Universal Robots URScript: test1.script

def unnamed():
  global _hidden_verificationVariable=0
  set_tcp(p[0.0,0.0,0.0,0.0,0.0,0.0])
  set_safety_mode_transition_hardness(1)
  set_gravity([0.0, 0.0, 9.82])
  set_tool_communication(False, 115200, 0, 1, 1.5, 3.5)
  set_tool_output_mode(0)
  set_tool_digital_output_mode(0, 1)
  set_tool_digital_output_mode(1, 1)
  set_tool_voltage(0)
  set_target_payload(0.000000, [0.000000, 0.000000, 0.000000], [0.000000, 0.000000, 0.000000, 0.000000, 0.000000, 0.000000])
  set_standard_analog_input_domain(0, 1)
  set_standard_analog_input_domain(1, 1)
  set_tool_analog_input_domain(0, 1)
  set_tool_analog_input_domain(1, 1)
  set_analog_outputdomain(0, 0)
  set_analog_outputdomain(1, 0)
  set_input_actions_to_default()
  # begin: URCap Installation Node
  #   Source: External Control, 1.0.5, FZI Research Center for Information Technology
  #   Type: External Control
  # end: URCap Installation Node
  step_count_bf1d607d_5cad_4ca6_951d_d38089d2c4e9 = 0.0
  thread Step_Counter_Thread_272bec76_1d24_4e5e_b286_867ec8d2c18c():
    while (True):
      step_count_bf1d607d_5cad_4ca6_951d_d38089d2c4e9 = step_count_bf1d607d_5cad_4ca6_951d_d38089d2c4e9 + 1.0
      sync()
    end
  end
  run Step_Counter_Thread_272bec76_1d24_4e5e_b286_867ec8d2c18c()
  global Waypoint_1_p=p[.365377612465, -.462828783151, .512939210108, -1.170877947002, 2.833532311999, .102825613587]
  global Waypoint_1_q=[-0.6912114986220512, -1.7813268732349261, -1.267368403083033, -1.6883155612163208, 1.667533326914021, 0.09468801413845322]
  global Waypoint_2_p=p[.000000000000, -.232900000168, 1.079399999952, -.000000000000, 2.221441469307, -2.221441468851]
  global Waypoint_2_q=[0.0, -1.5707963267948966, 0.0, -1.5707963267948974, 0.0, 0.0]
  global Waypoint_3_p=p[-.817200000000, -.232899999959, .062799999952, 1.570796327000, .000000000000, .000000000000]
  global Waypoint_3_q=[0.0, 0.0, 0.0, 0.0, 0.0, 0.0]
  while (True):
    $ 2 "Robot Program"
    $ 3 "MoveJ"
    $ 4 "Waypoint_1" "breakAfter"
    movej(Waypoint_1_q, a=1.3962634015954636, v=1.0471975511965976)
    $ 5 "Waypoint_2" "breakAfter"
    movej(Waypoint_2_q, a=1.3962634015954636, v=1.0471975511965976)
    $ 6 "Waypoint_3" "breakAfter"
    movej(Waypoint_3_q, a=1.3962634015954636, v=1.0471975511965976)
  end
end
